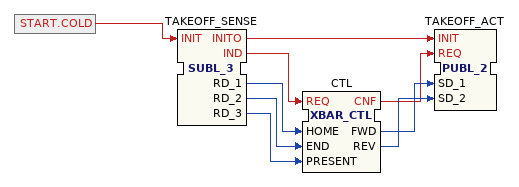
      FBS
        TAKEOFF_SENSE : SUBL_3;
        CTL : XBAR_CTL;
        TAKEOFF_ACT : PUBL_2;
      END_FBS
      EVENT_CONNECTIONS
        START.COLD TO TAKEOFF_SENSE.INIT;
        TAKEOFF_SENSE.INITO TO TAKEOFF_ACT.INIT;
        TAKEOFF_SENSE.IND TO CTL.REQ;
        CTL.CNF TO TAKEOFF_ACT.REQ;
      END_CONNECTIONS
      DATA_CONNECTIONS
        TAKEOFF_SENSE.RD_1 TO CTL.HOME;
        TAKEOFF_SENSE.RD_2 TO CTL.END;
        TAKEOFF_SENSE.RD_3 TO CTL.PRESENT;
        CTL.FWD TO TAKEOFF_ACT.SD_1;
        CTL.REV TO TAKEOFF_ACT.SD_2;
      END_CONNECTIONS
    END_RESOURCE
    DATA_CONNECTIONS
      3 TO SUPPLY_ACTUATORS.ROWS;
      3 TO DRILL_ACTUATORS.ROWS;
      3 TO SLIDE_ACTUATORS.ROWS;
      3 TO UNLOAD_ACTUATORS.ROWS;
      3 TO LOAD_ACTUATORS.ROWS;
      3 TO TAKEOFF_ACTUATORS.ROWS;
    END_CONNECTIONS
  END_DEVICE
  DATA_CONNECTIONS (* parameter values *)
    [100,100,375,360] TO CONTROL.BOUNDS;
    [6,2] TO CONTROL.GRID;
    [475,100,190,360] TO MODEL.BOUNDS;
  END_CONNECTIONS
END_SYSTEM
